FUNCTION_BLOCK E_CTU_CUSTOM
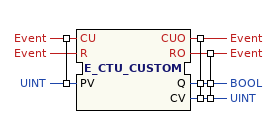
  EVENT_INPUT
    CU WITH PV;
    R;
  END_EVENT
  EVENT_OUTPUT
    CUO WITH Q, CV;
    RO WITH Q, CV;
  END_EVENT
  VAR_INPUT
    PV : UINT := 0;
  END_VAR
  VAR_OUTPUT
    Q : BOOL := FALSE;
    CV : UINT := 0;
  END_VAR
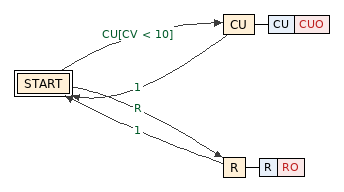
  EC_STATES
    START;
    CU : CU -> CUO;
    R : R -> RO;
  END_STATES
  EC_TRANSITIONS
    CU TO START := 1;
    START TO CU := CU[CV < 10];
    START TO R := R;
    R TO START := 1;
  END_TRANSITIONS
  ALGORITHM R IN ST:
CV := 0;
Q := FALSE;
  END_ALGORITHM
  ALGORITHM CU IN ST:
CV := CV + 1;
Q := (CV >= PV);
  END_ALGORITHM
END_FUNCTION_BLOCK
